Fanuc KAREL source: kt00168.KL

-- PROVISIONAL review KL for V1013-1; original PC SHA256 f1b94e292ec2a6436e41be84e8565f27f63a094947d6406f60c3680b97a31c4b
-- Incomplete behavior may be omitted. Consult companion uncertainty JSON. Do not deploy.
PROGRAM KT00168
%NOLOCKGROUP
VAR
  I1 : INTEGER
  OUT : REAL
-- UNRESOLVED_DECL H2 type=002017
BEGIN
  -- UNRESOLVED_PC offsets 5-16; opcodes 2E,23
  -- UNRESOLVED_PC offsets 21-35; opcodes 2E,22,9D,33,B4
  -- UNRESOLVED_PC offsets 40-63; opcodes 21,22,9D,33,B3,56,64,23
  -- UNRESOLVED_PC offsets 68-72; opcodes 7F
END KT00168
